// TwinCAT 3 PLC project PlcMain
// ProgramVersion: 3.1.4023.0
// libraries:
//   Tc2_MC2, * (Beckhoff Automation GmbH)
//   Tc2_SerialCom, * (Beckhoff Automation GmbH)
//   Tc2_Standard, * (Beckhoff Automation GmbH)
//   Tc2_System, * (Beckhoff Automation GmbH)
//   Tc3_Module, * (Beckhoff Automation GmbH)
// project tree:
//   DUTs/ State.TcDUT (not stored), StateCnv.TcDUT, StateDisp.TcDUT (not stored), StateHeat.TcDUT, StateMan.TcDUT (not stored), StateSeparator.TcDUT (not stored), StateTr.TcDUT (not stored), StateVe.TcDUT
//   GVLs/ GVL_SAFETY.TcGVL, GVL_VIS.TcGVL, IFC_HW.TcGVL, SerialComRFID.TcGVL, SerialComWaage.TcGVL
//   / PlcTask.TcTTO
//   POUs/ FB_Conveyor.TcPOU (not stored), FB_Dispenser.TcPOU, FB_FillLevel.TcPOU (not stored), FB_HeatingSystem.TcPOU (not stored), FB_ManipulatorAxis.TcPOU (not stored), FB_RFID.TcPOU (not stored), FB_Separator.TcPOU, FB_StatusLight.TcPOU, FB_TBlink.TcPOU, FB_Transport.TcPOU (not stored), FB_Waage.TcPOU (not stored), F_map.TcPOU (not stored), MAIN.TcPOU, PRG_CommRFID.TcPOU, PRG_CommWaage.TcPOU, PRG_Lab.TcPOU
// real-time tasks:
//   TASK PlcTask: cycle T#10ms, priority 20, ADS port 350
// motion (NC):
//   TASK NC-Task 1 SAF: cycle T#2ms, priority 4, ADS port 501
//   TASK NC-Task 1 SVB: cycle T#10ms, priority 8, ADS port 511
//   AXIS Conveyor (id 1)
//     Dynamic: AccelerationMaximum=700, DecelerationMaximum=700, Acceleration=400, Deceleration=400, Jerk=6000
//     Velo: SlowManual=10, FastManual=50, Maximum=50
//     OtherSettings: AllowMotionCmdToSlave=true
//     encoder EncType=4
//       EncPara: MaxCount=#x0000ffff
//     drive DrvType=23
//       Analog: VeloReferenz=50, TorqueSetpointScale=10, ScaleFactorActTorque=0.1
//       TimeComp: TaskDelayCycles=1
//     controller CtrType=1
//       CtrPara: PriorControlFactor=1
//         Observer: BandWidth=20
//   AXIS ManX (id 2)
//     Dynamic: AccelerationMaximum=1000, DecelerationMaximum=1000, Acceleration=1000, Deceleration=1000, Jerk=20160
//     Velo: SlowManual=10, FastManual=100, Maximum=280
//     OtherSettings: AllowMotionCmdToSlave=true
//     encoder EncType=4
//       EncPara: MaxCount=#x0000ffff
//     drive DrvType=24
//       Analog: VeloReferenz=320, TorqueSetpointScale=10, ScaleFactorActTorque=0.1
//       TimeComp: TaskDelayCycles=1
//     controller CtrType=1
//       CtrPara: PriorControlFactor=1
//         Observer: BandWidth=20
//   AXIS ManY (id 3)
//     Dynamic: AccelerationMaximum=1000, DecelerationMaximum=1000, Acceleration=1000, Deceleration=1000, Jerk=20160
//     Velo: SlowManual=10, FastManual=100, Maximum=280
//     OtherSettings: AllowMotionCmdToSlave=true
//     encoder EncType=4
//       EncPara: MaxCount=#x0000ffff
//     drive DrvType=24
//       Analog: VeloReferenz=320, TorqueSetpointScale=10, ScaleFactorActTorque=0.1
//       TimeComp: TaskDelayCycles=1
//     controller CtrType=1
//       CtrPara: PriorControlFactor=1
//         Observer: BandWidth=20
//   AXIS ManZ (id 4)
//     Dynamic: AccelerationMaximum=500, DecelerationMaximum=500, Acceleration=176.4, Deceleration=176.4, Jerk=1103.44
//     Velo: RefSearch=15, RefSync=15, SlowManual=15, FastManual=15, Maximum=60
//     OtherSettings: AllowMotionCmdToSlave=true, PulseDistancePos=10, PulseDistanceNeg=10
//     encoder EncType=4
//       EncPara: MaxCount=#x0000ffff
//     drive DrvType=24
//       Analog: VeloReferenz=254, TorqueSetpointScale=10, ScaleFactorActTorque=0.1
//       TimeComp: TaskDelayCycles=1
//     controller CtrType=1
//       CtrPara: PriorControlFactor=1
//         Observer: BandWidth=20
//   AXIS Disp1 (id 5)
//     Dynamic: AccelerationMaximum=3000, DecelerationMaximum=3000, Acceleration=2300, Deceleration=2300, Jerk=5290
//     Velo: Maximum=3600
//     OtherSettings: AllowMotionCmdToSlave=true
//     encoder EncType=4
//       EncPara: MaxCount=#x0000ffff
//     drive DrvType=24
//       Analog: VeloReferenz=3600, TorqueSetpointScale=10, ScaleFactorActTorque=0.1
//       TimeComp: TaskDelayCycles=1
//     controller CtrType=1
//       CtrPara: PriorControlFactor=1
//         Observer: BandWidth=20
//   AXIS Disp2 (id 6)
//     Dynamic: AccelerationMaximum=3000, DecelerationMaximum=3000, Acceleration=2300, Deceleration=2300, Jerk=5290
//     Velo: Maximum=3600
//     OtherSettings: AllowMotionCmdToSlave=true
//     encoder EncType=4
//       EncPara: MaxCount=#x0000ffff
//     drive DrvType=24
//       Analog: VeloReferenz=3600, TorqueSetpointScale=10, ScaleFactorActTorque=0.1
//       TimeComp: TaskDelayCycles=1
//     controller CtrType=1
//       CtrPara: PriorControlFactor=1
//         Observer: BandWidth=20
//   AXIS Disp3 (id 7)
//     Dynamic: AccelerationMaximum=3000, DecelerationMaximum=3000, Acceleration=2300, Deceleration=2300, Jerk=5290
//     Velo: Maximum=3600
//     OtherSettings: AllowMotionCmdToSlave=true
//     encoder EncType=4
//       EncPara: MaxCount=#x0000ffff
//     drive DrvType=24
//       Analog: VeloReferenz=3600, TorqueSetpointScale=10, ScaleFactorActTorque=0.1
//       TimeComp: TaskDelayCycles=1
//     controller CtrType=1
//       CtrPara: PriorControlFactor=1
//         Observer: BandWidth=20
//   AXIS ManGrip (id 8)
//     Dynamic: AccelerationMaximum=10, DecelerationMaximum=10, Acceleration=4.10666, Deceleration=4.10666, Jerk=7.80775
//     Velo: Maximum=4
//     OtherSettings: AllowMotionCmdToSlave=true
//     encoder EncType=4
//       EncPara: MaxCount=#x0000ffff
//     drive DrvType=24
//       Analog: VeloReferenz=17, TorqueSetpointScale=10, ScaleFactorActTorque=0.1
//       TimeComp: TaskDelayCycles=1
//     controller CtrType=1
//       CtrPara: PriorControlFactor=1
//         Observer: BandWidth=20
// I/O:
//   DEVICE Gerät 1 (EtherCAT Automation Protocol), AmsNetId 169.254.59.75.2.1
//     Box From Model (Subscriber)
//     Box To Model (Publisher)
// variable links:
//   NC-Task 1 SAF/Axes/Conveyor <-> Device 1 (EtherCAT Automation Protocol)/Box From Model (Subscriber)
//     Drive/Inputs/In/nState1 <-> DriveState/Inputs/VarData[0]
//     Enc/Inputs/In/nDataIn1[0] <-> DriveCounterValue/Inputs/VarData[0]
//   NC-Task 1 SAF/Axes/Conveyor <-> Device 1 (EtherCAT Automation Protocol)/Box To Model (Publisher)
//     Drive/Outputs/Out/nDataOut2[0] <-> DriveVelocity/Outputs/VarData[0]
//   NC-Task 1 SAF/Axes/Disp1 <-> Device 1 (EtherCAT Automation Protocol)/Box From Model (Subscriber)
//     Drive/Inputs/In/nState1 <-> DriveState/Inputs/VarData[1]
//     Enc/Inputs/In/nDataIn1[0] <-> DriveCounterValue/Inputs/VarData[1]
//   NC-Task 1 SAF/Axes/Disp1 <-> Device 1 (EtherCAT Automation Protocol)/Box To Model (Publisher)
//     Drive/Outputs/Out/nDataOut2[0] <-> DriveVelocity/Outputs/VarData[1]
//   NC-Task 1 SAF/Axes/Disp2 <-> Device 1 (EtherCAT Automation Protocol)/Box From Model (Subscriber)
//     Drive/Inputs/In/nState1 <-> DriveState/Inputs/VarData[2]
//     Enc/Inputs/In/nDataIn1[0] <-> DriveCounterValue/Inputs/VarData[2]
//   NC-Task 1 SAF/Axes/Disp2 <-> Device 1 (EtherCAT Automation Protocol)/Box To Model (Publisher)
//     Drive/Outputs/Out/nDataOut2[0] <-> DriveVelocity/Outputs/VarData[2]
//   NC-Task 1 SAF/Axes/Disp3 <-> Device 1 (EtherCAT Automation Protocol)/Box From Model (Subscriber)
//     Drive/Inputs/In/nState1 <-> DriveState/Inputs/VarData[3]
//     Enc/Inputs/In/nDataIn1[0] <-> DriveCounterValue/Inputs/VarData[3]
//   NC-Task 1 SAF/Axes/Disp3 <-> Device 1 (EtherCAT Automation Protocol)/Box To Model (Publisher)
//     Drive/Outputs/Out/nDataOut2[0] <-> DriveVelocity/Outputs/VarData[3]
//   NC-Task 1 SAF/Axes/ManGrip <-> Device 1 (EtherCAT Automation Protocol)/Box From Model (Subscriber)
//     Drive/Inputs/In/nState1 <-> DriveState/Inputs/VarData[7]
//     Enc/Inputs/In/nDataIn1[0] <-> DriveCounterValue/Inputs/VarData[7]
//   NC-Task 1 SAF/Axes/ManGrip <-> Device 1 (EtherCAT Automation Protocol)/Box To Model (Publisher)
//     Drive/Outputs/Out/nDataOut2[0] <-> DriveVelocity/Outputs/VarData[7]
//   NC-Task 1 SAF/Axes/ManX <-> Device 1 (EtherCAT Automation Protocol)/Box From Model (Subscriber)
//     Drive/Inputs/In/nState1 <-> DriveState/Inputs/VarData[4]
//     Enc/Inputs/In/nDataIn1[0] <-> DriveCounterValue/Inputs/VarData[4]
//   NC-Task 1 SAF/Axes/ManX <-> Device 1 (EtherCAT Automation Protocol)/Box To Model (Publisher)
//     Drive/Outputs/Out/nDataOut2[0] <-> DriveVelocity/Outputs/VarData[4]
//   NC-Task 1 SAF/Axes/ManY <-> Device 1 (EtherCAT Automation Protocol)/Box From Model (Subscriber)
//     Drive/Inputs/In/nState1 <-> DriveState/Inputs/VarData[5]
//     Enc/Inputs/In/nDataIn1[0] <-> DriveCounterValue/Inputs/VarData[5]
//   NC-Task 1 SAF/Axes/ManY <-> Device 1 (EtherCAT Automation Protocol)/Box To Model (Publisher)
//     Drive/Outputs/Out/nDataOut2[0] <-> DriveVelocity/Outputs/VarData[5]
//   NC-Task 1 SAF/Axes/ManZ <-> Device 1 (EtherCAT Automation Protocol)/Box From Model (Subscriber)
//     Drive/Inputs/In/nState1 <-> DriveState/Inputs/VarData[6]
//     Enc/Inputs/In/nDataIn1[0] <-> DriveCounterValue/Inputs/VarData[6]
//   NC-Task 1 SAF/Axes/ManZ <-> Device 1 (EtherCAT Automation Protocol)/Box To Model (Publisher)
//     Drive/Outputs/Out/nDataOut2[0] <-> DriveVelocity/Outputs/VarData[6]
//   PlcMain/PlcMain Instance <-> Device 1 (EtherCAT Automation Protocol)/Box From Model (Subscriber)
//     PlcTask Inputs/IFC_HW.BandSens{1..4} <-> BandSens/Inputs/VarData[{0..3}]  (4 links)
//     PlcTask Inputs/IFC_HW.EinzelSens1 <-> VereinzSens/Inputs/VarData[0]
//     PlcTask Inputs/IFC_HW.EinzelSens2 <-> VereinzSens/Inputs/VarData[1]
//     PlcTask Inputs/IFC_HW.EinzelSens3 <-> VereinzSens/Inputs/VarData[2]
//   PlcMain/PlcMain Instance <-> Device 1 (EtherCAT Automation Protocol)/Box To Model (Publisher)
//     PlcTask Outputs/IFC_HW.BandHub1 <-> BandHub/Outputs/VarData[0]
//     PlcTask Outputs/IFC_HW.BandHub2 <-> BandHub/Outputs/VarData[1]
//     PlcTask Outputs/IFC_HW.BandHub3 <-> BandHub/Outputs/VarData[2]
//     PlcTask Outputs/IFC_HW.R1AKT1 <-> VereinzHub/Outputs/VarData[0,0]
//     PlcTask Outputs/IFC_HW.R1AKT2 <-> VereinzHub/Outputs/VarData[1,0]
//     PlcTask Outputs/IFC_HW.R2AKT1 <-> VereinzHub/Outputs/VarData[0,1]
//     PlcTask Outputs/IFC_HW.R2AKT2 <-> VereinzHub/Outputs/VarData[1,1]
//   PlcMain/PlcMain Instance <-> NC-Task 1 SAF/Axes/Conveyor
//     PlcTask Inputs/IFC_HW.BandMotor.NcToPlc <-> Outputs/ToPlc
//     PlcTask Outputs/IFC_HW.BandMotor.PlcToNc <-> Inputs/FromPlc
//   PlcMain/PlcMain Instance <-> NC-Task 1 SAF/Axes/Disp1
//     PlcTask Inputs/IFC_HW.BandExtruder1.NcToPlc <-> Outputs/ToPlc
//     PlcTask Outputs/IFC_HW.BandExtruder1.PlcToNc <-> Inputs/FromPlc
//   PlcMain/PlcMain Instance <-> NC-Task 1 SAF/Axes/Disp2
//     PlcTask Inputs/IFC_HW.BandExtruder2.NcToPlc <-> Outputs/ToPlc
//     PlcTask Outputs/IFC_HW.BandExtruder2.PlcToNc <-> Inputs/FromPlc
//   PlcMain/PlcMain Instance <-> NC-Task 1 SAF/Axes/Disp3
//     PlcTask Inputs/IFC_HW.BandExtruder3.NcToPlc <-> Outputs/ToPlc
//     PlcTask Outputs/IFC_HW.BandExtruder3.PlcToNc <-> Inputs/FromPlc
//   PlcMain/PlcMain Instance <-> NC-Task 1 SAF/Axes/ManGrip
//     PlcTask Inputs/IFC_HW.ManAchseGrip.NcToPlc <-> Outputs/ToPlc
//     PlcTask Outputs/IFC_HW.ManAchseGrip.PlcToNc <-> Inputs/FromPlc
//   PlcMain/PlcMain Instance <-> NC-Task 1 SAF/Axes/ManX
//     PlcTask Inputs/IFC_HW.ManAchseX.NcToPlc <-> Outputs/ToPlc
//     PlcTask Outputs/IFC_HW.ManAchseX.PlcToNc <-> Inputs/FromPlc
//   PlcMain/PlcMain Instance <-> NC-Task 1 SAF/Axes/ManY
//     PlcTask Inputs/IFC_HW.ManAchseY.NcToPlc <-> Outputs/ToPlc
//     PlcTask Outputs/IFC_HW.ManAchseY.PlcToNc <-> Inputs/FromPlc
//   PlcMain/PlcMain Instance <-> NC-Task 1 SAF/Axes/ManZ
//     PlcTask Inputs/IFC_HW.ManAchseZ.NcToPlc <-> Outputs/ToPlc
//     PlcTask Outputs/IFC_HW.ManAchseZ.PlcToNc <-> Inputs/FromPlc

CONFIGURATION PlcMain
    RESOURCE PLC ON TwinCAT3
        TASK PlcTask(INTERVAL := T#10ms, PRIORITY := 20);
        PROGRAM PRG_Lab WITH PlcTask : PRG_Lab;
    END_RESOURCE
END_CONFIGURATION

// ---- DUTs/StateCnv.TcDUT
{attribute 'qualified_only'}
{attribute 'strict'}
TYPE StateCnv :
(
	Off,
	Reset,
	Power,
	Ready,
	Moving
);
END_TYPE

// ---- DUTs/StateHeat.TcDUT
{attribute 'qualified_only'}
{attribute 'strict'}
TYPE StateHeat :
(
	Off,
	Init,
	Ready,
	Heat,
	Hold,
	Done
);
END_TYPE

// ---- DUTs/StateVe.TcDUT
{attribute 'qualified_only'}
{attribute 'strict'}
TYPE StateVe :
(
	Off,
	Fill,
	Idle,
	Eject,
	Done,
	Error
);
END_TYPE

// ---- GVLs/GVL_SAFETY.TcGVL
{attribute 'qualified_only'}
VAR_GLOBAL
	safebLightBarrierOK AT%I* 	: BOOL; // Light barrier OK
	safebEmergencyStopOK AT%I* 	: BOOL; // Emergency stop OK
	safebDoorLockedOK AT%I* 	: BOOL; // Safety door locked OK
		
	bAcknowledge_Button AT%I* 	: BOOL;	// Input acknowledge button
	bBetrieb_Button AT%I* 		: BOOL; // Input start factory button
	bBetrieb_Out AT%Q* 			: BOOL;
	
	safeLockDoor AT%Q*			: BOOL; // Safety lock door
	safebAcknowledge AT%Q* 		: BOOL; // Safety acknowledge
	safebErrAck AT%Q* 			: BOOL;	// Safety error acknowledge
	safeOverruled AT%Q*			: BOOL; // Safety overruled
	safebSafeRun AT%Q* 			: BOOL := TRUE; // Safety run

END_VAR

// ---- GVLs/GVL_VIS.TcGVL
{attribute 'qualified_only'}
VAR_GLOBAL
	bSetup 		: BOOL; // Start setup mode
	bProduction : BOOL; // Start production mode
	
	bStartFactoryHMI : BOOL; // Start factory button HMI
	bAcknowledgeHMI  : BOOL; // Acknowledge button HMI
	bStorageHMI		 : BOOL; // Overrule button HMI
	
	bActuator1	: BOOL; // Start actuator 1
	bActuator2	: BOOL; // Start actuator 2
	bRFID		: BOOL; // Start RFID
	bConveyor 	: BOOL; // Start Conveyor
	bDispenser1 : BOOL;	// Start dispenser 1
	bDispenser2 : BOOL; // Start dispenser 2
	bDispenser3 : BOOL;	// Start dispenser 3
	sFilling1 : STRING; // Input value dispenser 1
	sFilling2 : STRING;	// Input value dispenser 2
	sFilling3 : STRING;	// Input value dispenser 3
	
	bHeating : BOOL; 		// Start Heating button
	rHeating : REAL := 0; 	// Value of heating (0-5V)
	
	bAxisX : BOOL;		// Start x axis button
	bAxisY : BOOL;		// Start y axis button
	bAxisZ : BOOL;		// Start z axis button
	bAxisG : BOOL;		// Start gripper axis button 
	sAxisX : STRING;	// Input value x axis
	sAxisY : STRING;	// Input value y axis
	sAxisZ : STRING;	// Input value z axis
	sAxisG : STRING;	// Input value gripper axis
	
	TSens1	: REAL; // Heating block temperature 1
	TSens2	: REAL; // Heating block temperature 2
	TSens	: REAL; // Heating block tamperature
	                
	GEmpty 	: BOOL; // Error granulate empty
	FullSt	: BOOL; // Error full storage
	WrongB	: BOOL; // Error wrong bottle
	NoB		: BOOL; // Error no bottle
	
END_VAR

// ---- GVLs/IFC_HW.TcGVL
// In dieser GVL werden alle Variablen deklariert die auf die realen Klemmen zugreifen
VAR_GLOBAL
	// Errors 
		NoBottle			: BOOL := FALSE; // Keine Flasche vorhanden
		WrongBottle			: BOOL := FALSE; // Flasche falsch gedreht oder falsche Flasche
		StorageFull			: BOOL := FALSE; // Lager abgefüllte Flaschen voll
		GranulateEmpty		: BOOL := FALSE; // Füllstand Granulat zu gering
		
	// Station Statusampel	
		AmpelRot 	AT%Q* 	: BOOL;		// Signal-LED Rot
		AmpelGelb 	AT%Q* 	: BOOL;		// Signal-LED Gelb
		AmpelGrun 	AT%Q* 	: BOOL;		// Signal-LED Grun
			
	// Station Vereinzelung
		EinzelSens1 AT%I*	: BOOL;			// Separation Sensor 1
		EinzelSens2 AT%I*	: BOOL;			// Separation Sensor 2
		EinzelSens3 AT%I*	: BOOL;			// Separation Sensor 3
		R1AKT1 	AT%Q* 		: BOOL;			// Relais 1 Aktor 1
		R2AKT1 	AT%Q* 		: BOOL;			// Relais 2 Aktor 1
		R1AKT2 	AT%Q* 		: BOOL;			// Relais 1 Aktor 2
		R2AKT2 	AT%Q* 		: BOOL;			// Relais 2 Aktor 2
	
	// Station Forderband
		BandSens1 AT %I*	: BOOL;		// Forderband Sensor 1
		BandSens2 AT %I*	: BOOL;		// Forderband Sensor 2
		BandSens3 AT %I*	: BOOL;		// Forderband Sensor 3
		BandSens4 AT %I*	: BOOL;		// Forderband Sensor 4
		BandHub1 AT %Q*		: BOOL;		// Forderband Hubmagnet 1
		BandHub2 AT %Q*		: BOOL;		// Forderband Hubmagnet 1
		BandHub3 AT %Q*		: BOOL;		// Forderband Hubmagnet 1
		BandExtruder1 		: AXIS_REF;	// Forderband NC-Achse Dosiereinheit 1
		BandExtruder2 		: AXIS_REF;	// Forderband NC-Achse Dosiereinheit 2
		BandExtruder3 		: AXIS_REF;	// Forderband NC-Achse Dosiereinheit 3
		BandMotor 			: AXIS_REF;	// Forderband NC-Achse Band
		
		BandFullmenge1		: INT := 5;	// in Gramm
		BandFullmenge2		: INT := 7;	// in Gramm
		BandFullmenge3		: INT := 3;	// in Gramm
		
	//Füllstandsüberwachung
		FillSens1 AT%I*	: UINT;			// Füllstandssensor 1
		FillSens2 AT%I*	: UINT;			// Füllstandssensor 2
		FillSens3 AT%I*	: UINT;			// Füllstandssensor 3
		FillLevelPercent1	: REAL;		// Füllstand 1 in %
		FillLevelGramm1		: REAL;		// Füllstand i in g
		FillLevelPercent2	: REAL;		// Füllstand 2 in %
		FillLevelGramm2		: REAL;		// Füllstand 2 in g
		FillLevelPercent3	: REAL;		// Füllstand 3 in %
		FillLevelGramm3		: REAL;		// Füllstand 3 in g
		
		MaxFillLevel 	: REAL := 375;	// Kalibrierter Füllstand für 10% * 10
		
	// Station Waage
		WaageNachricht		: STRING;	// Nachricht von Wagezelle (fur virtuelle Inbetriebnahme notig)
		WaageNull			: BOOL;		// TARA Waage
		WaageMesswert		: INT;		// Messwert der Waage
		
	// Station Behalteridentifikation
		IdSensorTrager			: BOOL;		// Sensor bei Erkennung eines Datentrager
		IdNachricht				: STRING;	// Nachricht von RFID-System (fur virtuelle Inbetriebnahme notig)
		Seriennummer			: STRING;	// Seriennummer RFID-Tag
		
	//Temperierstation
		Ventilator1 AT %Q*	: BOOL;		// Ventilator 1
		Ventilator2 AT %Q*	: BOOL;		// Ventilator 2
		Ventilator3 AT %Q*	: BOOL;		// Ventilator 3
		TempSens1 AT%I*		: UINT;		// Temperatursensor 1
		TempSens2 AT%I*		: UINT;		// Temperatursensor 2
		Heizpatrone AT%Q*	: UINT;		// Heizpatronen
		MaxTemp				: UINT := 5500;		// in °C * 100
		
	// Station Manipulator
		ManEndX AT%I* 		: BOOL := TRUE;		// Manipulator min Endschalter Achse x
		ManEndY AT%I* 		: BOOL := TRUE;		// Manipulator min Endschalter Achse y
		ManEndZ AT%I* 		: BOOL := TRUE;		// Manipulator min Endschalter Achse z
		ManEndGrip AT%I* 	: BOOL := TRUE;		// Manipulator min Endschalter Achse Gripper
		ManEndX2 AT%I* 		: BOOL := TRUE;		// Manipulator max Endschalter Achse x
		ManEndY2 AT%I* 		: BOOL := TRUE;		// Manipulator max Endschalter Achse y
		ManEndZ2 AT%I* 		: BOOL := TRUE;		// Manipulator max Endschalter Achse z
		ManEndGrip2 AT%I* 	: BOOL := TRUE;		// Manipulator max Endschalter Achse Gripper
		Brake	AT%Q*		: BOOL := FALSE;	// Bremse Achse z
		
		ManAchseX			: AXIS_REF;			// Manipulator NC-Achse x
		ManAchseY			: AXIS_REF;			// Manipulator NC-Achse y
		ManAchseZ			: AXIS_REF;			// Manipulator NC-Achse z
		ManAchseGrip		: AXIS_REF; 		// Manipulator NC-Achse Gripper
END_VAR

// ---- GVLs/SerialComRFID.TcGVL
VAR_GLOBAL
	ELDataIn_RFID AT %I* : EL6inData22B;
	ELDataOut_RFID AT %Q* : EL6outData22B;

	RecRFID : ReceiveString;
	
	RxBufferRFID : ComBuffer;
	TxBufferRFID : ComBuffer;
	
	ErrorFastRFID : BOOL;
	
END_VAR

// ---- GVLs/SerialComWaage.TcGVL
VAR_GLOBAL
	ELDataIn_Waage AT %I* : EL6inData22B;
	ELDataOut_Waage AT %Q* : EL6outData22B;
	
	RecWaage : ReceiveString;
	TxWaage : SendString;
	
	RxBufferWaage : ComBuffer;
	TxBufferWaage : ComBuffer;
	
	ErrorFastWaage : BOOL;
	
END_VAR

// ---- POUs/PRG_Lab.TcPOU
PROGRAM PRG_Lab
VAR
	fbStatusLight : FB_StatusLight;
	
	fbSeparator : FB_Separator;
	
	fbRFID : FB_RFID;
	
	fbConveyor : FB_Conveyor;
	
	fbFillLevel1 : FB_FillLevel;
	fbFillLevel2 : FB_FillLevel;
	fbFillLevel3 : FB_FillLevel;
	
	fbDisp1 : FB_Dispenser;
	fbDisp2 : FB_Dispenser;
	fbDisp3 : FB_Dispenser;
	
	fbManX  : FB_ManipulatorAxis;
	fbManY  : FB_ManipulatorAxis;
	fbManZ  : FB_ManipulatorAxis;
	fbManGrip 	: FB_ManipulatorAxis;
	
	fbWaage : FB_Waage;
	
	fbHeating : FB_HeatingSystem;
	
	nState : INT := 0;
	nCount : INT := 0;
	
	timer : TON;
END_VAR

fbStatusLight(
	bRed=> IFC_HW.AmpelRot,
	bYellow=> IFC_HW.AmpelGelb,
	bGreen=> IFC_HW.AmpelGrun);

fbSeparator(
	bSensor1:= IFC_HW.EinzelSens1, 
	bSensor2:= IFC_HW.EinzelSens2, 
	bR1AKT1=> IFC_HW.R1AKT1, 
	bR1AKT2=> IFC_HW.R1AKT2,
	bR2AKT1=> IFC_HW.R2AKT1, 
	bR2AKT2=> IFC_HW.R2AKT2,
	bNoBottle=> IFC_HW.NoBottle,	
	bWrongBottle=> IFC_HW.WrongBottle);
	
fbRFID( 
	sSeriennummer=> IFC_HW.IdNachricht);

fbConveyor(
	ax:= IFC_HW.BandMotor);

fbFillLevel1(
	nLevelIn:= IFC_HW.FillSens1,
	nMaxLevel:= IFC_HW.MaxFillLevel,
	nLevelPercent=> IFC_HW.FillLevelPercent1,
	nLevelGramm=> IFC_HW.FillLevelGramm1);
fbFillLevel2(
	nLevelIn:= IFC_HW.FillSens2,
	nMaxLevel:= IFC_HW.MaxFillLevel,
	nLevelPercent=> IFC_HW.FillLevelPercent2,
	nLevelGramm=> IFC_HW.FillLevelGramm2);
fbFillLevel3(
	nLevelIn:= IFC_HW.FillSens3,
	nMaxLevel:= IFC_HW.MaxFillLevel,
	nLevelPercent=> IFC_HW.FillLevelPercent3,
	nLevelGramm=> IFC_HW.FillLevelGramm3);
	
fbDisp1(
	ax:= IFC_HW.BandExtruder1);
fbDisp2(
	ax:= IFC_HW.BandExtruder2);
fbDisp3(
	ax:= IFC_HW.BandExtruder3);

fbManX(
	aAchse:= IFC_HW.ManAchseX,
	bEndSchalterMin:=IFC_HW.ManEndX,
	bEndSchalterMax:=IFC_HW.ManEndX2);
fbManY(
	aAchse:= IFC_HW.ManAchseY,
	bEndSchalterMin:=IFC_HW.ManEndY,
	bEndSchalterMax:=IFC_HW.ManEndY2);
fbManZ(
	aAchse:= IFC_HW.ManAchseZ,
	bEndSchalterMin:=IFC_HW.ManEndZ,
	bEndSchalterMax:=IFC_HW.ManEndZ2);
	
fbManGrip(
	aAchse:= IFC_HW.ManAchseGrip,
	bEndSchalterMin:=IFC_HW.ManEndGrip,
	bEndSchalterMax:=IFC_HW.ManEndGrip2);
	
fbWaage(
	bNullsetzen:= IFC_HW.WaageNull,
	iMesswert=> IFC_HW.WaageMesswert);
	
fbHeating(
	nMaxTemp:= IFC_HW.MaxTemp,
	nTemp:= (IFC_HW.TempSens1 + IFC_HW.TempSens2)/2,
	bVentilator1=> IFC_HW.Ventilator1,
	bVentilator2=> IFC_HW.Ventilator2,
	bVentilator3=> IFC_HW.Ventilator3,
	nHeizpatrone=> IFC_HW.Heizpatrone);	
	
CASE nState OF
0: // Off
	fbStatusLight.eStatus := State.Off;
	fbSeparator.bEnable := FALSE;
	fbConveyor.bEnable := FALSE;
	fbDisp1.bEnable := FALSE;
	fbDisp2.bEnable := FALSE;
	fbDisp3.bEnable := FALSE;
	fbHeating.bEnable := FALSE;
	fbManX.bEnable := FALSE;
	fbManY.bEnable := FALSE;
	fbManZ.bEnable := FALSE;
	fbManGrip.bEnable := FALSE;
	
	nState := nState + 1;
	
1: // Turn on
	fbStatusLight.eStatus := State.Busy;
	fbSeparator.bEnable := TRUE;
	fbConveyor.bEnable := TRUE;
	fbDisp1.bEnable := TRUE;
	fbDisp2.bEnable := TRUE;
	fbDisp3.bEnable := TRUE;
	fbHeating.bEnable := TRUE;
	IFC_HW.Brake := TRUE;
	fbManZ.bEnable := TRUE;
	IF fbManZ.eOutState = State.Ready THEN
		IFC_HW.Brake := FALSE;
		fbManX.bEnable := TRUE;
		fbManY.bEnable := TRUE;
		fbManGrip.bEnable := TRUE;
	END_IF
	
	IF fbSeparator.eStatus = State.Ready
		AND fbConveyor.eStatus = State.Ready
		AND fbDisp1.eStatus = State.Ready
		AND fbDisp2.eStatus = State.Ready
		AND fbDisp3.eStatus = State.Ready
		AND fbHeating.eStatus = State.Ready
		AND fbManX.eOutState = State.Ready
		AND fbManY.eOutState = State.Ready
		AND fbManGrip.eOutState = State.Ready THEN
		nState := nState + 1;
	END_IF

2: // check error
	IF nCount >= 4 THEN
		fbStatusLight.eStatus := State.Error;
		IFC_HW.StorageFull := TRUE;
		IF GVL_SAFETY.safeOverruled AND GVL_SAFETY.bAcknowledge_Button THEN
			IFC_HW.StorageFull := FALSE;
			GVL_SAFETY.safeOverruled := FALSE;
			nCount := 0;
			nState := nState + 1;
		END_IF
	ELSIF  NOT IFC_HW.EinzelSens2 AND NOT IFC_HW.EinzelSens3 THEN
		fbStatusLight.eStatus := State.Error;
		IFC_HW.NoBottle := TRUE;
		IF GVL_SAFETY.bAcknowledge_Button THEN
			IFC_HW.NoBottle := FALSE;
			nState := 1;
		END_IF
	ELSIF (NOT IFC_HW.EinzelSens2 AND IFC_HW.EinzelSens3) OR (IFC_HW.EinzelSens2 AND IFC_HW.EinzelSens3)THEN
		fbStatusLight.eStatus := State.Error;
		IFC_HW.WrongBottle := TRUE;
		IF GVL_SAFETY.bAcknowledge_Button THEN
			IFC_HW.WrongBottle := FALSE;
			nState := 1;
		END_IF
	ELSIF IFC_HW.FillLevelPercent1 < 5 OR IFC_HW.FillLevelPercent2 < 5 OR IFC_HW.FillLevelPercent3 < 5 THEN
		fbStatusLight.eStatus := State.Error;
		IFC_HW.GranulateEmpty := TRUE;
		IF GVL_SAFETY.bAcknowledge_Button THEN
			IFC_HW.GranulateEmpty := FALSE;
			nState := 1;
		END_IF
	ELSE
		nState := nState + 1;
	END_IF
	
3: // All systems ready
	fbStatusLight.eStatus := State.Ready;
	
	IF (GVL_SAFETY.bBetrieb_Button OR GVL_VIS.bStartFactoryHMI) AND NOT GVL_SAFETY.safeOverruled THEN
		GVL_SAFETY.bBetrieb_Button := FALSE; // reset
		nState := nState + 1;
	END_IF
	
4: // read RFID
	fbStatusLight.eStatus := State.Busy;
	//fbRFID.bSensorTrager := TRUE;
	
	//IF fbRFID.bFertig THEN
		//fbRFID.bSensorTrager := FALSE;
		nState := nState + 1;
	//END_IF
	
5: // separate container
	fbSeparator.bExecute := TRUE;
	
	IF fbSeparator.eStatus = State.Done THEN
		fbSeparator.bExecute := FALSE;
		nState := nState + 1;
	END_IF
	
6: // turn on conveyor and wait for container to arrive at BandSens1
	fbConveyor.eDirection := MC_Direction.MC_Positive_Direction;
	fbConveyor.nVel := 40;
	fbConveyor.bExecute := TRUE;
	
	IF IFC_HW.BandSens1 THEN
		timer(IN := TRUE, PT := T#500MS);
		IF timer.Q THEN
			fbConveyor.bExecute := FALSE;
			timer(IN := FALSE);
			nState := nState + 1;
		END_IF
	END_IF
	
7: // fill container from first dispenser
	fbDisp1.nDispenseGrams := IFC_HW.BandFullmenge1;
	fbDisp1.bExecute := TRUE;
	
	IF fbDisp1.eStatus = State.Done THEN
		fbDisp1.bExecute := FALSE;
		nState := nState + 1;
	END_IF
	
8: // continue conveyor to second dispenser (BandSens2)
	fbConveyor.eDirection := MC_Direction.MC_Positive_Direction;
	fbConveyor.nVel := 40;
	
	fbConveyor.bExecute := TRUE;
	
	IFC_HW.BandHub1 := TRUE;
	
	IF IFC_HW.BandSens2 THEN
		timer(IN := TRUE, PT := T#500MS);
		IF timer.Q THEN
			fbConveyor.bExecute := FALSE;
			IFC_HW.BandHub1 := FALSE;
			timer(IN := FALSE);
			nState := nState + 1;
		END_IF
	END_IF
	
9: // fill container from second dispenser
	fbDisp2.nDispenseGrams := IFC_HW.BandFullmenge2;
	fbDisp2.bExecute := TRUE;
	
	IF fbDisp2.eStatus = State.Done THEN
		fbDisp2.bExecute := FALSE;
		nState := nState + 1;
	END_IF
	
10: // continue conveyor to third dispenser (BandSens3)
	fbConveyor.eDirection := MC_Direction.MC_Positive_Direction;
	fbConveyor.nVel := 40;
	fbConveyor.bExecute := TRUE;
	
	IFC_HW.BandHub2 := TRUE;
	
	IF IFC_HW.BandSens3 THEN
		timer(IN := TRUE, PT := T#500MS);
		IF timer.Q THEN
			fbConveyor.bExecute := FALSE;
			IFC_HW.BandHub2 := FALSE;
			timer(IN := FALSE);
			nState := nState + 1;
		END_IF
	END_IF
	
11: // fill container from second dispenser
	fbDisp3.nDispenseGrams := IFC_HW.BandFullmenge3;
	fbDisp3.bExecute := TRUE;
	
	IF fbDisp3.eStatus = State.Done THEN
		fbDisp3.bExecute := FALSE;
		nState := nState + 1;
	END_IF
	
12: // continue conveyor to end of line (BandSens4)
	fbConveyor.eDirection := MC_Direction.MC_Positive_Direction;
	fbConveyor.nVel := 40;
	fbConveyor.bExecute := TRUE;
	
	IFC_HW.BandHub3 := TRUE;
	
	IF IFC_HW.BandSens4 THEN
		timer(IN := TRUE, PT := T#500MS);
		IF timer.Q THEN
			fbConveyor.bExecute := FALSE;
			IFC_HW.BandHub3 := FALSE;
			timer(IN := FALSE);
			nState := nState + 1;
		END_IF
	END_IF

13: // open Gripper
	fbManGrip.fVelocity := 3;	
	fbManGrip.fPosition := 6;
	
	fbManGrip.bExecute := TRUE;	
	
	IF fbManGrip.eOutState = State.Done THEN
		fbManGrip.bExecute := FALSE;
		nState := nState + 1;
	END_IF
		
14: // goto container x, y
	fbManX.fVelocity := 30;
	fbManY.fVelocity := 30;
	
	fbManX.fPosition := 31;
	fbManY.fPosition := 145;
	
	fbManX.bExecute := TRUE;
	fbManY.bExecute := TRUE;
	
	IF fbManX.eOutState = State.Done AND fbManY.eOutState = State.Done THEN
		fbManX.bExecute := FALSE;
		fbManY.bExecute := FALSE;
		nState := nState + 1;
	END_IF
	
15: // goto container z	
	fbManZ.fVelocity := 30;
	
	fbManZ.fPosition := 132;
	
	IFC_HW.Brake := TRUE;
	fbManZ.bExecute := TRUE;
	
	IF fbManZ.eOutState = State.Done THEN
		fbManZ.bExecute := FALSE;
		IFC_HW.Brake := FALSE;
		nState := nState + 1;
	END_IF

16: // close Gripper
	fbManGrip.fPosition := 8.5;
	
	fbManGrip.bExecute := TRUE;	
	
	IF fbManGrip.eOutState = State.Done THEN
		fbManGrip.bExecute := FALSE;
		nState := nState + 1;
	END_IF

17: // move Z UP
	fbManZ.fPosition := 70;

	IFC_HW.Brake := TRUE;
	fbManZ.bExecute := TRUE;	
	
	IF fbManZ.eOutState = State.Done THEN
		fbManZ.bExecute := FALSE;
		IFC_HW.Brake := FALSE;
		nState := nState + 1;
	END_IF

18: // goto scale x, y
	fbManX.fPosition := 37;
	fbManY.fPosition := 7;
	
	fbManX.bExecute := TRUE;
	fbManY.bExecute := TRUE;
	
	IF fbManX.eOutState = State.Done AND fbManY.eOutState = State.Done THEN
		fbManX.bExecute := FALSE;
		fbManY.bExecute := FALSE;
		nState := nState + 1;
	END_IF

19: // set scale to zero	
	//IFC_HW.WaageNull := TRUE;
	
	//IF fBWaage.iMesswert = 0 THEN
		nState := nState + 1;
	//END_IF

20: // goto scale z	
	fbManZ.fPosition := 132.5;
	
	IFC_HW.Brake := TRUE;
	fbManZ.bExecute := TRUE;
	
	IF fbManZ.eOutState = State.Done THEN
		fbManZ.bExecute := FALSE;
		IFC_HW.Brake := FALSE;
		nState := nState + 1;
	END_IF
	
21: // open Gripper		
	fbManGrip.fPosition := 6;
	
	fbManGrip.bExecute := TRUE;
	
	IF fbManGrip.eOutState = State.Done THEN
		fbManGrip.bExecute := FALSE;
		nState := nState + 1;
	END_IF
	
22: // scale 
	nState := nState + 1;
	
23: // close Gripper
	fbManGrip.fPosition := 8.5;	
	
	fbManGrip.bExecute := TRUE;	
	
	IF fbManGrip.eOutState = State.Done THEN
		fbManGrip.bExecute := FALSE;
		nState := nState + 1;
	END_IF

24: // move Z UP	
	fbManZ.fPosition := 70;
	
	IFC_HW.Brake := TRUE;
	fbManZ.bExecute := TRUE;
	
	IF fbManZ.eOutState = State.Done THEN
		fbManZ.bExecute := FALSE;
		IFC_HW.Brake := FALSE;
		nState := nState + 1;
	END_IF
	
25: // goto heating x, y
	fbManX.fPosition := 220.5;
	fbManY.fPosition := 6;
	
	fbManX.bExecute := TRUE;
	fbManY.bExecute := TRUE;
	
	IF fbManX.eOutState = State.Done AND fbManY.eOutState = State.Done THEN
		fbManX.bExecute := FALSE;
		fbManY.bExecute := FALSE;
		nState := nState + 1;
	END_IF

26: // goto heating z	
	fbManZ.fPosition := 180;
	
	IFC_HW.Brake := TRUE;
	fbManZ.bExecute := TRUE;
	
	IF fbManZ.eOutState = State.Done THEN
		fbManZ.bExecute := FALSE;
		IFC_HW.Brake := FALSE;
		nState := nState + 1;
	END_IF

27: // open Gripper	
	fbManGrip.fPosition := 6;
	
	fbManGrip.bExecute := TRUE;	
	
	IF fbManGrip.eOutState = State.Done THEN
		fbManGrip.bExecute := FALSE;
		nState := nState + 1;
	END_IF
	
28: // heating 
	fbHeating.bExecute := TRUE;
	
	IF fbHeating.eStatus = State.Done THEN
		fbHeating.bExecute := FALSE;
		nState := nState + 1;
	END_IF

29: // close Gripper
	fbManGrip.fPosition := 8.5;	
	
	fbManGrip.bExecute := TRUE;	
	
	IF fbManGrip.eOutState = State.Done THEN
		fbManGrip.bExecute := FALSE;
		nState := nState + 1;
	END_IF

30: // move Z UP	
	fbManZ.fPosition := 70;
	
	IFC_HW.Brake := TRUE;
	fbManZ.bExecute := TRUE;
	
	IF fbManZ.eOutState = State.Done THEN
		fbManZ.bExecute := FALSE;
		IFC_HW.Brake := FALSE;
		nState := nState + 1;
	END_IF

31: // goto storage x, y
	CASE nCount OF		
	0: // storage 1
		fbManX.fPosition := 110.5;
	1: // storage 2
		fbManX.fPosition := 161.5;
	2: // storage 3
		fbManX.fPosition := 212.5;
	3: // storage 4
		fbManX.fPosition := 263;	
	END_CASE
	
	fbManY.fPosition := 138;
	
	fbManX.bExecute := TRUE;
	fbManY.bExecute := TRUE;
	
	IF fbManX.eOutState = State.Done AND fbManY.eOutState = State.Done THEN
		fbManX.bExecute := FALSE;
		fbManY.bExecute := FALSE;
		nCount := nCount + 1;
		nState := nState + 1;
	END_IF

32: // goto storage z	
	fbManZ.fPosition := 128;
	
	IFC_HW.Brake := TRUE;
	fbManZ.bExecute := TRUE;
	
	IF fbManZ.eOutState = State.Done THEN
		fbManZ.bExecute := FALSE;
		IFC_HW.Brake := FALSE;
		nState := nState + 1;
	END_IF	
	
33: // open Gripper		
	fbManGrip.fPosition := 6;
	
	fbManGrip.bExecute := TRUE;
	
	IF fbManGrip.eOutState = State.Done THEN
		fbManGrip.bExecute := FALSE;
		nState := nState + 1;
	END_IF
	
34: // move Z UP
	fbManZ.fPosition := 80;
	
	IFC_HW.Brake := TRUE;
	fbManZ.bExecute := TRUE;
	
	IF fbManZ.eOutState = State.Done THEN
		fbManZ.bExecute := FALSE;
		IFC_HW.Brake := FALSE;
		nState := nState + 1;
	END_IF
	
35: // goto container x, y
	fbManX.fPosition := 31;
	fbManY.fPosition := 145;
	
	fbManX.bExecute := TRUE;
	fbManY.bExecute := TRUE;
	
	IF fbManX.eOutState = State.Done AND fbManY.eOutState = State.Done THEN
		fbManX.bExecute := FALSE;
		fbManY.bExecute := FALSE;
		nState := nState + 1;
	END_IF
	
36: // Done
	fbStatusLight.eStatus := State.Done;
	
	timer(IN := TRUE, PT := T#3000MS);
	
	IF timer.Q THEN
		timer(IN := FALSE);
		nState := 1;
	END_IF
	
END_CASE

END_PROGRAM

// ---- POUs/FB_StatusLight.TcPOU
FUNCTION_BLOCK FB_StatusLight
VAR_INPUT
	eStatus : State;
END_VAR
VAR_OUTPUT
	bRed : BOOL := FALSE;
	bYellow : BOOL := FALSE;
	bGreen : BOOL := FALSE;
END_VAR
VAR
	fbBlink : FB_TBlink;
END_VAR

fbBlink(IN:=TRUE, PT:=T#500MS);

CASE eStatus OF
State.Off:
	bRed := TRUE;
	bYellow := FALSE;
	bGreen := FALSE;
State.Busy:
	bRed := FALSE;
	bYellow := TRUE;
	bGreen := FALSE;
State.Ready:
	bRed := FALSE;
	bYellow := FALSE;
	bGreen := TRUE;
State.Done:
	bRed := FALSE;
	bYellow := FALSE;
	bGreen := fbBlink.Q;
State.Error:
	bRed := fbBlink.Q;
	bYellow := FALSE;
	bGreen := FALSE;
State.Setup:
	bRed := FALSE;
	bYellow := fbBlink.Q;
	bGreen := fbBlink.Q;;
END_CASE

END_FUNCTION_BLOCK

// ---- POUs/FB_TBlink.TcPOU
FUNCTION_BLOCK FB_TBlink
VAR_INPUT
	IN: BOOL;
	PT: TIME;
END_VAR
VAR_OUTPUT
	Q: BOOL;
END_VAR
VAR
	fbTimer: TP;
END_VAR

fbTimer(IN:=IN AND NOT fbTimer.Q, PT:=PT);

IF IN AND fbTimer.ET < PT/2 THEN
	Q := TRUE;
ELSE
	Q := FALSE;
END_IF

END_FUNCTION_BLOCK

// ---- POUs/FB_Separator.TcPOU
FUNCTION_BLOCK FB_Separator
VAR_INPUT
	bEnable : BOOL; 	// start/stops the functionblock
	bExecute: BOOL; 	// Ejects 1 flask if true
	bErrorReset: BOOL;	//Reset Error 
	
	bSensor1 : BOOL; //Hardware Sensor 1
	bSensor2 : BOOL; //Hardware Sensor 2
	bSensor3 : BOOL; //Hardware Sensor 3
END_VAR
VAR_OUTPUT
	bR1AKT1 : BOOL; //Relais 1 Aktor 1 (Schieber oben)
	bR2AKT1 : BOOL; //Relais 2 Aktor 1
	bR1AKT2 : BOOL; //Relais 1 Aktor 2 (Schieber unten)
	bR2AKT2 : BOOL; //Relais 2 Aktor 2
	
	bNoBottle		: BOOL;		//Keine Flasche vorhanden
	bWrongBottle	: BOOL; //Falsche oder gedrehte Flasche vorhanden
	
	eStatus : State := State.Off;
END_VAR
VAR
	timer : TON; //Timer to make sure, that the flask has cleared the slope
	eState : StateSeparator := StateSeparator.Off;
END_VAR

CASE eState OF
StateSeparator.Off:
	eStatus := State.Off;
	bR1AKT1 := TRUE;	//Eingefahren oben
	bR2AKT1 := FALSE;	//Eingefahren oben
	
	bR1AKT2 := FALSE;	//Eingefahren unten
	bR2AKT2 := TRUE;	//Eingefahren unten

	IF bEnable	THEN
		eState := StateSeparator.Init;
	END_IF
	
StateSeparator.Init:
	
	eStatus := State.Busy; //Beschaeftigt Signallampe

	bR1AKT1 := FALSE; //Ausgefahren oben
	bR2AKT1 := TRUE;
	
	bR1AKT2 := FALSE; //Eingefahren unten
	bR2AKT2 := TRUE;

	
	IF bSensor1 THEN
		eState := StateSeparator.Init_Wait;	//Zustandswechsel sobald Sensor Flasche zwischen Schiebern sieht
	END_IF	
	
StateSeparator.Init_Wait:
	timer(IN := TRUE, PT := T#1000MS); //Timer wartet bis Flasche sicher zum Stehen kommt
	
	IF timer.Q THEN
		timer(IN := FALSE);
		eState := StateSeparator.Ready; //Zustand Ready nach Timer
	END_IF
	
StateSeparator.Ready:
	eStatus := State.Ready; //Zustand Ready Signallampe

	bR1AKT1 := TRUE;	//Eingefahren oben
	bR2AKT1 := FALSE;	//Eingefahren oben
	
	bR1AKT2 := FALSE;	//Eingefahren unten
	bR2AKT2 := TRUE;	//Eingefahren unten
	
	IF bExecute THEN
		eState := StateSeparator.Eject_Wait_1; //Auswerfen sobald Exceute TRUE
	END_IF

StateSeparator.Eject_Wait_1:	// Warten bis Schieber oben ganz geschlossen ist
		eStatus := State.Busy; //Zustand Busy Signallampe
	
		timer(IN := TRUE, PT := T#2500MS); //Timer auf 2,5 S eingestellt
	
	IF timer.Q THEN
		timer(IN := FALSE);
		eState := StateSeparator.Eject; //Zustand bereit nach Timer
	END_IF
	
StateSeparator.Eject:	//Auswerfen der unteren Flasche
	bR1AKT2 := TRUE;	//Lässt Flaschen auf Band ab durch Öffnen des unteren Schiebers
	bR2AKT2 := FALSE;
	
	IF NOT bSensor1 THEN
		eState := StateSeparator.Eject_Wait_2; 
	END_IF
	
StateSeparator.Eject_Wait_2:	// Warten bis Flasche durch Förderband weit genug von Schieber wegtransportiert
	eStatus := State.Done;
	timer(IN := TRUE, PT := T#4000MS); //Timer auf 4 S eingestellt
	
	IF timer.Q THEN
		timer(IN := FALSE);
		eState := StateSeparator.Done_Wait; 
	END_IF 
	
StateSeparator.Done_Wait: // Schließen des unteren Schiebers und Warten bis komplettt geschlossen
	bR1AKT2 := FALSE;	//Eingefahren unten
	bR2AKT2 := TRUE;	//Eingefahren unten
	
	timer(IN := TRUE, PT := T#3000MS); //Timer wartet bis Schieber geschlossen ist
	
	IF timer.Q THEN
		timer(IN := FALSE);
		eState := StateSeparator.Done; 
	END_IF	
	
StateSeparator.Done:	//Vereinzelungsvorgang abgeschlossen
	
	IF NOT bExecute THEN
		eState := StateSeparator.Init;
	END_IF

END_CASE

END_FUNCTION_BLOCK

// ---- POUs/FB_Dispenser.TcPOU
// Das ist die Musterlosung zur Steuerung einer Dosiereinheit.
// Library TC2_MC2 ist notig.

FUNCTION_BLOCK FB_Dispenser
	VAR_INPUT
		bEnable					: BOOL;
		bExecute				: BOOL;
		nDispenseGrams			: INT := 1;		// Gewunschte Menge in Gramm
	END_VAR

	VAR_OUTPUT
		eStatus	: State := State.Off;
	END_VAR
	
	VAR_IN_OUT
		ax		: AXIS_REF; 			// Referenz auf die NC-Achse
	END_VAR

	VAR
		// Fur NC-Achse notig
		fbReset			: MC_Reset;
		fbPower			: MC_Power;
		fbMove			: MC_MoveRelative;
		
		// Parameter
		nVelocity			: INT := 720;		// Grad pro Sekunde
		fGramPerRev			: REAL := 0.245;		// Skalierung auf Gramm pro ganzer Umdrehung (360 Grad)
		
		// Working variables
		eState				: StateDisp;		// Status der Zustandsmaschine
		bAxPower			: BOOL;
		bAxMove				: BOOL;
END_VAR
	
// ----- Ende der Definition. Hier folgt der Code ------


// update axis
ax.ReadStatus();

// call NC FBs
fbReset(
	Axis:= ax);
fbPower(
	Axis:= ax, 
	Enable:= bAxPower, 
	Enable_Positive:= bAxPower, 
	Enable_Negative:= bAxPower, 
	Override:= 100);
fbMove(
	Axis:=ax,
	Execute:=bAxMove,
	Velocity:=nVelocity,
	Distance:= nDispenseGrams *360 / fGramPerRev);
	
	

IF NOT bEnable THEN
	eState := StateDisp.Off;
END_IF

CASE eState OF
StateDisp.Off:
	eStatus := State.Off;
	bAxMove := FALSE;
	bAxPower := FALSE;
	
	IF bEnable THEN
		eState := StateDisp.Reset;
	END_IF
StateDisp.Reset:
	eStatus := State.Busy;
	fbReset.Execute := TRUE;
	IF fbReset.Done THEN
		fbReset.Execute := FALSE;
		eState := StateDisp.PowerUp;
	END_IF
StateDisp.PowerUp:
	eStatus := State.Busy;
	bAxPower := TRUE;
	IF fbPower.Status THEN
		eState := StateDisp.Idle;
	END_IF
StateDisp.Idle:
	eStatus := State.Ready;
	bAxMove := FALSE;

	IF bExecute THEN
		eState := StateDisp.Dispensing;
	END_IF
StateDisp.Dispensing:
	eStatus := State.Busy;
	bAxMove := TRUE;
	
	IF fbMove.Done THEN
		eState := StateDisp.Done;
	END_IF
StateDisp.Done:
	eStatus := State.Done;
	bAxMove := FALSE;
	
	IF NOT bExecute THEN
		eState := StateDisp.Idle;
	END_IF
END_CASE

END_FUNCTION_BLOCK

// ---- POUs/MAIN.TcPOU
PROGRAM MAIN
VAR
	
END_VAR



GVL_SAFETY.safebAcknowledge := GVL_SAFETY.bAcknowledge_Button OR GVL_VIS.bAcknowledgeHMI;
GVL_SAFETY.bBetrieb_Out := GVL_SAFETY.bBetrieb_Button OR GVL_VIS.bStartFactoryHMI;

GVL_VIS.TSens1 := IFC_HW.TempSens1/100;
GVL_VIS.TSens2 := IFC_HW.TempSens2/100;
GVL_VIS.TSens := (GVL_VIS.TSens1+GVL_VIS.TSens2)/2;
	
GVL_VIS.GEmpty := NOT IFC_HW.GranulateEmpty;
GVL_VIS.FullSt := NOT IFC_HW.StorageFull;
GVL_VIS.WrongB := NOT IFC_HW.WrongBottle;
GVL_VIS.NoB := NOT IFC_HW.NoBottle;


IF GVL_SAFETY.safebEmergencyStopOK AND GVL_SAFETY.safebLightBarrierOK AND GVL_SAFETY.safebDoorLockedOK THEN
	IF GVL_VIS.bSetup THEN
		PRG_Setup();
	ELSIF GVL_VIS.bProduction THEN
		PRG_Lab();
	END_IF	
END_IF

END_PROGRAM

// ---- POUs/PRG_CommRFID.TcPOU
PROGRAM PRG_CommRFID
	VAR
		ControllerRFID : SerialLineControl;
	END_VAR

ControllerRFID(
	Mode:= SERIALLINEMODE_EL6_22B, 
	pComIn:= ADR(ELDataIn_RFID), 
	pComOut:= ADR(ELDataOut_RFID), 
	SizeComIn:= TO_UINT( SIZEOF(ELDataIn_RFID)), 
	Error=> ErrorFastRFID, 
	ErrorID=> , 
	TxBuffer:= TxBufferRFID, 
	RxBuffer:= RxBufferRFID);

END_PROGRAM

// ---- POUs/PRG_CommWaage.TcPOU
PROGRAM PRG_CommWaage
	VAR
		ControllerWaage : SerialLineControl;
		nCount : DINT := 0;
END_VAR

ControllerWaage(
	Mode:= SERIALLINEMODE_EL6_22B, 
	pComIn:= ADR(ELDataIn_Waage), 
	pComOut:= ADR(ELDataOut_Waage), 
	SizeComIn:= TO_UINT( SIZEOF(ELDataIn_Waage)), 
	Error=> ErrorFastWaage, 
	ErrorID=> , 
	TxBuffer:= TxBufferWaage, 
	RxBuffer:= RxBufferWaage);
	
	nCount := nCount + 1;

END_PROGRAM
